PROGRAM Rotina019
VAR
	status: INT;
	
	posicaoAtual: STRING;
	envialog: STRING;
	
	fbTimeVentila: ton;
	fbTimeAqueci: ton;
	
END_VAR

fbTimeVentila();
fbTimeAqueci();

CASE status OF

0:
IF gvl_p.arrStatusEstufas[0].start AND STRING_TO_DT(gvl.progInicio[0]) <= systemtime_to_dt(gvl.fbGetLocalSystemTime.systemTime)  THEN
	status:= 5;
	
	gvl.bstartchart019:= TRUE;
	gvl_p.zona1setpt_019:= gvl_p.arrStatusEstufas[0].tempSeca;
	gvl_p.zona2setpt_019:= gvl_p.arrStatusEstufas[0].tempSeca;
	gvl.liga_ventilacao_019:= TRUE;
	fbTimeVentila(in:= TRUE, pt:=T#1S);

///// GERADOR DE LOG -------------------------------------------------------------

envialog:= 'Inicializando Programação ESTUFA 019';
gvl.logRegister19:= envialog;

	gvl_p.etapa_process[0] := 'Inicializando';
	
ELSE
	status:= 0;
	IF gvl_p.arrStatusEstufas[0].start THEN
		gvl_p.etapa_process[0] := gvl.progInicio[0];
	END_IF
END_IF

5:
IF fbTimeVentila.Q THEN
	status:= 10;
	gvl.liga_ventilacao_019:=FALSE;
	fbTimeVentila(in:= FALSE);
ELSE
	status:= 5;
END_IF

10:
IF gvl.ventilacao_Ligada_019 THEN
	status:= 15;
	
	gvl.liga_aquecimento_019:= TRUE;
	fbTimeAqueci(in:= TRUE, pt:= T#1S);
	
///// GERADOR DE LOG -------------------------------------------------------------

envialog:= 'Aquecendo ESTUFA 019';
gvl.logRegister19:= envialog;
	
	gvl_p.etapa_process[0] := 'Aquecendo';
	
ELSE
	status:= 10;
END_IF

15:
IF fbTimeAqueci.Q THEN
	status:= 20;
	
	gvl.liga_aquecimento_019:= FALSE;
	fbTimeAqueci(in:=false);
ELSE
	status:= 15;
END_IF

20:
IF gvl.zona1atual_019 >= gvl_p.zona1setpt_019 THEN
	status:= 30;
	
gvl.progInicio[0]:= DT_TO_STRING(gvl.somaTempo);
	
///// CALCULAR FIM DA SECAGEM E DA ARMAZENAGEM --------------------------------------------------------------------------------
gvl_p.arrStatusEstufas[0].inicioSecagem := STRING_TO_DT(gvl.progInicio[0]);
gvl_p.arrStatusEstufas[0].fimSecagem := STRING_TO_DT(gvl.progInicio[0]) + gvl_p.arrStatusEstufas[0].tempoSecagem;
gvl_P.arrStatusEstufas[0].prevFimSeca := gvl_p.arrStatusEstufas[0].fimSecagem;
gvl_p.arrStatusEstufas[0].fimArmazenagem := gvl_p.arrStatusEstufas[0].fimSecagem + gvl_p.arrStatusEstufas[0].tempoArmazenagem ;

///// IMPRIMIR A HORA E A DATA DO INICIO DA SECAGEM ---------------------------------------------------------------------------
gvl_p.arrStatusEstufas[0].statusInicioSecagem := '';
gvl_p.arrStatusEstufas[0].statusInicioSecagem := concat(gvl_p.arrStatusEstufas[0].statusInicioSecagem,gvl.hora);
gvl_p.arrStatusEstufas[0].statusInicioSecagem := concat(gvl_p.arrStatusEstufas[0].statusInicioSecagem,':');
gvl_p.arrStatusEstufas[0].statusInicioSecagem := concat(gvl_p.arrStatusEstufas[0].statusInicioSecagem,gvl.minuto);
gvl_p.arrStatusEstufas[0].statusInicioSecagem := concat(gvl_p.arrStatusEstufas[0].statusInicioSecagem,' ');
gvl_p.arrStatusEstufas[0].statusInicioSecagem := concat(gvl_p.arrStatusEstufas[0].statusInicioSecagem,gvl.dia);
gvl_p.arrStatusEstufas[0].statusInicioSecagem := concat(gvl_p.arrStatusEstufas[0].statusInicioSecagem,'/');
gvl_p.arrStatusEstufas[0].statusInicioSecagem := concat(gvl_p.arrStatusEstufas[0].statusInicioSecagem,gvl.mes);
gvl_p.arrStatusEstufas[0].statusInicioSecagem := concat(gvl_p.arrStatusEstufas[0].statusInicioSecagem,'/');
gvl_p.arrStatusEstufas[0].statusInicioSecagem := concat(gvl_p.arrStatusEstufas[0].statusInicioSecagem,gvl.ano);

//--------------------REATOR------------------------------------

IF gravarConfigPosicao_Reator.bGravarConfigPosicao_Reator THEN
	gvl_p.arrStatusEstufas[0].inicioReator := '';
	gvl_p.arrStatusEstufas[0].inicioReator := concat(gvl_p.arrStatusEstufas[0].inicioReator,gvl.hora);
	gvl_p.arrStatusEstufas[0].inicioReator := concat(gvl_p.arrStatusEstufas[0].inicioReator,':');
	gvl_p.arrStatusEstufas[0].inicioReator := concat(gvl_p.arrStatusEstufas[0].inicioReator,gvl.minuto);
	gvl_p.arrStatusEstufas[0].inicioReator := concat(gvl_p.arrStatusEstufas[0].inicioReator,' ');
	gvl_p.arrStatusEstufas[0].inicioReator := concat(gvl_p.arrStatusEstufas[0].inicioReator,gvl.dia);
	gvl_p.arrStatusEstufas[0].inicioReator := concat(gvl_p.arrStatusEstufas[0].inicioReator,'/');
	gvl_p.arrStatusEstufas[0].inicioReator := concat(gvl_p.arrStatusEstufas[0].inicioReator,gvl.mes);
	gvl_p.arrStatusEstufas[0].inicioReator := concat(gvl_p.arrStatusEstufas[0].inicioReator,'/');
	gvl_P.arrStatusEstufas[0].inicioReator := concat(gvl_p.arrStatusEstufas[0].inicioReator,gvl.ano);
END_IF

///// DECOMPOR A VARIAVEL FIM DA SECAGEM -----------------------------------------------------------------------------------------------
gvl_p.arrStatusEstufas[0].diaSec := MID(STR:= DT_TO_STRING(gvl_p.arrStatusEstufas[0].fimSecagem) , LEN:= 2, POS:=12);
gvl_p.arrStatusEstufas[0].mesSec := MID(STR:= DT_TO_STRING(gvl_p.arrStatusEstufas[0].fimSecagem), LEN:= 2, POS:=9);
gvl_p.arrStatusEstufas[0].anoSec := MID(STR:= DT_TO_STRING(gvl_p.arrStatusEstufas[0].fimSecagem), LEN:= 2, POS:=6);
gvl_p.arrStatusEstufas[0].horaSec := MID(STR:= DT_TO_STRING(gvl_p.arrStatusEstufas[0].fimSecagem), LEN:= 2, POS:=15);
gvl_p.arrStatusEstufas[0].minutoSec := MID(STR:= DT_TO_STRING(gvl_p.arrStatusEstufas[0].fimSecagem), LEN:= 2, POS:=18);

///// IMPRIMIR A HORA E A DATA DO FIM DA SECAGEM --------------------------------------------------------------------------------------------------------
gvl_p.arrStatusEstufas[0].statusFimSecagem := '';
gvl_p.arrStatusEstufas[0].statusFimSecagem := concat(gvl_p.arrStatusEstufas[0].statusFimSecagem,gvl_p.arrStatusEstufas[0].horaSec);
gvl_p.arrStatusEstufas[0].statusFimSecagem := concat(gvl_p.arrStatusEstufas[0].statusFimSecagem,':');
gvl_p.arrStatusEstufas[0].statusFimSecagem := concat(gvl_p.arrStatusEstufas[0].statusFimSecagem,gvl_p.arrStatusEstufas[0].minutoSec);
gvl_p.arrStatusEstufas[0].statusFimSecagem := concat(gvl_p.arrStatusEstufas[0].statusFimSecagem,' ');
gvl_p.arrStatusEstufas[0].statusFimSecagem := concat(gvl_p.arrStatusEstufas[0].statusFimSecagem,gvl_p.arrStatusEstufas[0].diaSec);
gvl_p.arrStatusEstufas[0].statusFimSecagem := concat(gvl_p.arrStatusEstufas[0].statusFimSecagem,'/');
gvl_p.arrStatusEstufas[0].statusFimSecagem := concat(gvl_p.arrStatusEstufas[0].statusFimSecagem,gvl_p.arrStatusEstufas[0].mesSec);
gvl_p.arrStatusEstufas[0].statusFimSecagem := concat(gvl_p.arrStatusEstufas[0].statusFimSecagem,'/');
gvl_p.arrStatusEstufas[0].statusFimSecagem := concat(gvl_p.arrStatusEstufas[0].statusFimSecagem,gvl_p.arrStatusEstufas[0].anoSec);

///// DECOMPOR A VARIAVEL FIM DA ARMAZENAGEM -------------------------------------------------------------------------------------------
gvl_p.arrStatusEstufas[0].diaArm := MID(STR:= DT_TO_STRING(gvl_p.arrStatusEstufas[0].fimArmazenagem) , LEN:= 2, POS:=12);
gvl_p.arrStatusEstufas[0].mesArm := MID(STR:= DT_TO_STRING(gvl_p.arrStatusEstufas[0].fimArmazenagem), LEN:= 2, POS:=9);
gvl_p.arrStatusEstufas[0].anoArm := MID(STR:= DT_TO_STRING(gvl_P.arrStatusEstufas[0].fimArmazenagem), LEN:= 2, POS:=6);
gvl_p.arrStatusEstufas[0].horaArm := MID(STR:= DT_TO_STRING(gvl_P.arrStatusEstufas[0].fimArmazenagem), LEN:= 2, POS:=15);
gvl_p.arrStatusEstufas[0].minutoArm := MID(STR:= DT_TO_STRING(gvl_p.arrStatusEstufas[0].fimArmazenagem), LEN:= 2, POS:=18);

///// IMPRIMIR A HORA E A DATA DO FIM DA ARMAZENAGEM -----------------------------------------------------------------------------------------------------------
gvl_p.arrStatusEstufas[0].statusFimArmazenagem := '';
gvl_p.arrStatusEstufas[0].statusFimArmazenagem := concat(gvl_p.arrStatusEstufas[0].statusFimArmazenagem,gvl_p.arrStatusEstufas[0].horaArm);
gvl_p.arrStatusEstufas[0].statusFimArmazenagem := concat(gvl_p.arrStatusEstufas[0].statusFimArmazenagem,':');
gvl_p.arrStatusEstufas[0].statusFimArmazenagem := concat(gvl_p.arrStatusEstufas[0].statusFimArmazenagem,gvl_p.arrStatusEstufas[0].minutoArm);
gvl_p.arrStatusEstufas[0].statusFimArmazenagem := concat(gvl_p.arrStatusEstufas[0].statusFimArmazenagem,' ');
gvl_p.arrStatusEstufas[0].statusFimArmazenagem := concat(gvl_p.arrStatusEstufas[0].statusFimArmazenagem,gvl_p.arrStatusEstufas[0].diaArm);
gvl_p.arrStatusEstufas[0].statusFimArmazenagem := concat(gvl_p.arrStatusEstufas[0].statusFimArmazenagem,'/');
gvl_p.arrStatusEstufas[0].statusFimArmazenagem := concat(gvl_p.arrStatusEstufas[0].statusFimArmazenagem,gvl_p.arrStatusEstufas[0].mesArm);
gvl_p.arrStatusEstufas[0].statusFimArmazenagem := concat(gvl_p.arrStatusEstufas[0].statusFimArmazenagem,'/');
gvl_p.arrStatusEstufas[0].statusFimArmazenagem := concat(gvl_p.arrStatusEstufas[0].statusFimArmazenagem,gvl_p.arrStatusEstufas[0].anoArm);

//gvl.permanencia[1]:= DT_TO_TIME(gvl_p.arrStatusEstufas[0].inicioSecagem);
///// GERADOR DE LOG -------------------------------------------------------------

envialog:= 'Secagem Iniciada ESTUFA 019';
gvl.logRegister19:= envialog;

gvl_p.etapa_process[0] := 'Secagem';

ELSE
	status:= 20;
END_IF

30:
IF gvl_p.arrStatusEstufas[0].prevFimSeca = systemtime_to_dt(gvl.fbGetLocalSystemTime.systemTime) THEN
	status:= 40;
	
	gvl_p.zona1setpt_019:= gvl_p.arrStatusEstufas[0].tempArm;
	gvl_p.zona2setpt_019:= gvl_p.arrStatusEstufas[0].tempArm;
	
///// GERADOR DE LOG -------------------------------------------------------------
envialog:= 'Armazenagem Iniciada ESTUFA 019';
gvl.logRegister19:= envialog;
	
gvl_p.etapa_process[0] := 'Armazenagem';

ELSE
	status:= 30;
END_IF

40:
IF gvl_p.arrStatusEstufas[0].fimArmazenagem = systemtime_to_dt(gvl.fbGetLocalSystemTime.systemTime) THEN
	status:= 50;
	
	gvl_p.arrStatusEstufas[0].start:= FALSE;
	gvl.bstartchart019:= FALSE;
	gvl.desl_aquecimento_019:= TRUE;
	fbTimeAqueci(in:=TRUE, pt:=T#1S);
	
	gvl_p.etapa_process[0] := '';
	
	gvl_p.arrStatusEstufas[0].statusInicioSecagem := '';
	gvl_p.arrStatusEstufas[0].inicioReator := '';
	gvl_p.arrStatusEstufas[0].statusFimSecagem := '';
	gvl_p.arrStatusEstufas[0].statusFimArmazenagem := '';
	gvl_p.arrStatusEstufas[0].fimSecagem:= DT#1970-1-1-0:0:0;
	gvl.endArm19:= T#0S;
	gvl.endSeca19:= T#0S;
	
	
///// GERADOR DE LOG -------------------------------------------------------------
envialog:= 'Programação Finalizada ESTUFA 019';
gvl.logRegister19:= envialog;

gvl_p.etapa_process[0]:= '';

ELSE
	status:= 40;
END_IF

45:
IF gvl_p.arrStatusEstufas[0].start THEN
status:= 50;
	
	gvl_p.arrStatusEstufas[0].start:= FALSE;
	gvl.bstartchart019:= FALSE;
	gvl.desl_aquecimento_019:= TRUE;
	fbTimeAqueci(in:=TRUE, pt:=T#1S);
	
	gvl_p.etapa_process[0] := '';
	
	gvl_p.arrStatusEstufas[0].statusInicioSecagem := '';
	gvl_p.arrStatusEstufas[0].inicioReator := '';
	gvl_p.arrStatusEstufas[0].statusFimSecagem := '';
	gvl_p.arrStatusEstufas[0].statusFimArmazenagem := '';
	gvl_p.arrStatusEstufas[0].fimSecagem:= DT#1970-1-1-0:0:0;
	gvl.endArm19:= T#0S;
	gvl.endSeca19:= T#0S;
	
///// GERADOR DE LOG -------------------------------------------------------------
envialog:= 'Programação Finalizada ESTUFA 019';
gvl.logRegister19:= envialog;

gvl_p.etapa_process[0]:= '';

ELSE
	status:= 45;
END_IF

50:
IF fbTimeAqueci.Q THEN
	status:= 0;
	
	gvl.desl_aquecimento_019:= FALSE;
	fbTimeAqueci(in:= FALSE);
	
ELSE
	status:= 50;
END_IF
END_CASE

END_PROGRAM

(* stored: Version 1.1.0.1, ProductVersion 3.1.4024.12
   POU Rotina019: Id {293bb9a6-b170-476f-abd8-825629ec8de0}, SpecialFunc None *)
